{attribute 'qualified_only'}
{attribute 'strict'}
TYPE E_StewartMode :
(
	SETTLED := 0,
	NEUTRAL,
	SIMULATION,
	GENERATOR,
	FILE
) USINT ;
END_TYPE

(* stored: Version 1.1.0.1, ProductVersion 3.1.4022.18
   DUT E_StewartMode: Id {e8e86642-4f9a-45ef-b209-c304e7ac55fa} *)
